{attribute 'qualified_only'}
{attribute 'strict'}
TYPE E_CYLINDER_Name :
(
	CLAMP				:=1,
	GATE				:=2,
	REJECT				:=3,
	ADDITIONAL_REJECT	:=4,  {text 'change to ADDIT'}
	FIRST_PUSHER		:=5,
	SECOND_PUSHER		:=6

);
END_TYPE

(* stored: Version 1.1.0.1
   DUT E_CYLINDER_Name: Id {7687e0d0-2fd8-41d7-8800-f65181b12042} *)
